(* Logix 5000 project; controller ktc_lab12 vendor 1 type 14 code 150 rev 30.11; software revision 30.00 *)

TASK MainTask (continuous, watchdog 500 ms) : MainProgram

MODULES
   Local : vendor 1 type 14 code 150 (Compact 0, rev 30.11)
      Counters : Embedded (Compact 3, rev 1.1, Output RPI 20 ms)
      Discrete_IO : Embedded (Compact 1, rev 3.1, Output RPI 20 ms)
      Analog_IO : Embedded (Compact 2, rev 1.1, Output RPI 80 ms)
END_MODULES

PROGRAM MainProgram   (* main routine MainRoutine *)
VAR
   array1 : DINT[10] := ([1] := 1, [2] := 2, [3] := 4, [4] := 8, [5] := 1, [6] := 3, [7] := 7, [8] := 15);   // count
   CONTROL1 : CONTROL := (LEN := 8, POS := 1, EN := 1);
   OUTPUT1 : DINT := 1;
   T4_1 : TIMER := (PRE := 1000, ACC := 141, EN := 1, TT := 1);   // DELY
END_VAR

ROUTINE MainRoutine   (* ladder *)
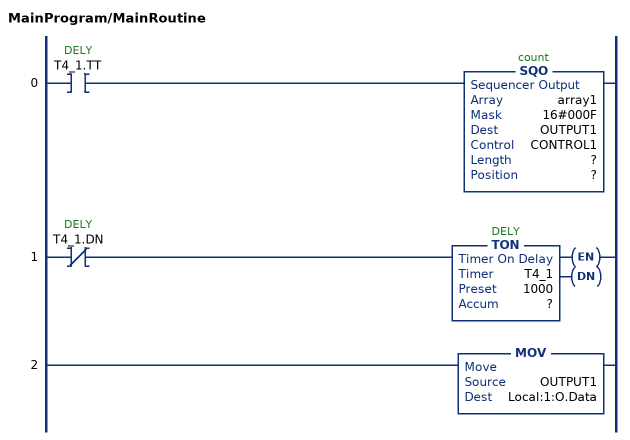
   0: XIC(T4_1.TT)SQO(array1,16#000F,OUTPUT1,CONTROL1,?,?);
   1: XIO(T4_1.DN)TON(T4_1,?,?);
   2: MOV(OUTPUT1,Local:1:O.Data);
END_ROUTINE
END_PROGRAM
